RoboDK station: RoboDK.rdk

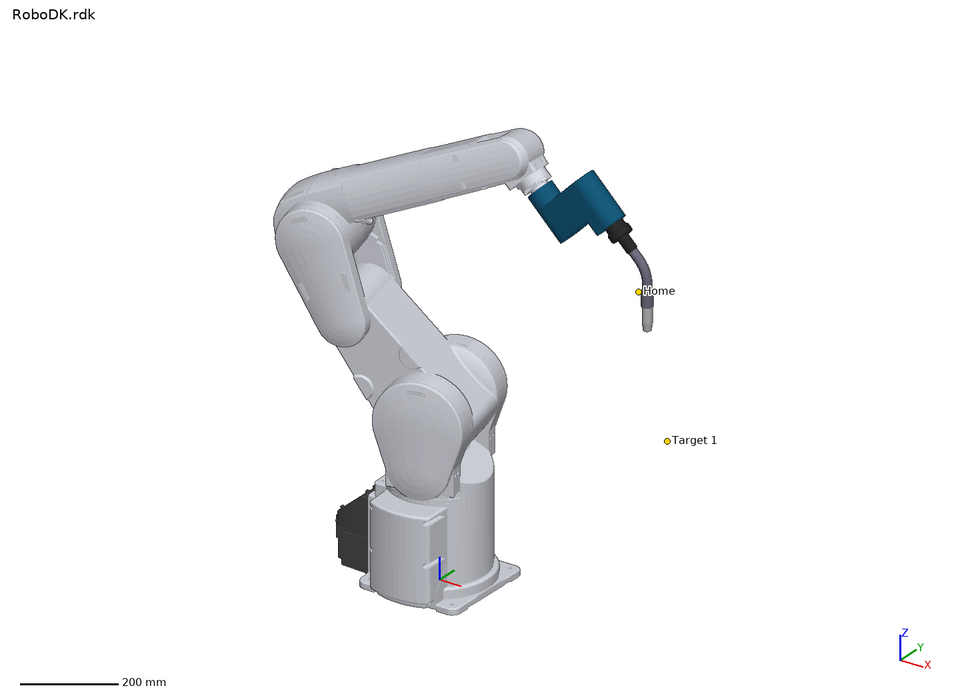
[picture v0: the station drawn from its stored meshes, robots at their saved joint values, targets as dots, program paths as lines]
Station 123. Poses are relative to the parent item; angles as X-Y-Z fixed-axis rotations.
  - frame Mitsubishi RV-7FL Base at (0, 0, 0) mm
    - robot Mitsubishi RV-7FL: 6 axes, payload 7 kg, reach 908 mm, repeatability 0.02 mm, weight 67 kg
        modified DH rows (alpha deg, a mm, theta deg, d mm): 0, 0, 0, 400; -90, 0, -90, 0; 0, 435, -90, 0; -90, 50, 0, 470; 90, 0, 0, 0; -90, 0, 180, 85
        joint limits [-240, -110, 0, -200, -120, -360] to [240, 130, 162, 200, 120, 360]; home [0, 0, 90, 0, 0, 0]; saved at [13.161, -34.303, 100.935, -9.903, 69.415, 12.901]
      - tool Weld gun, TCP at (-4, 0, 371.3) mm, rotated rx 0 ry 45 rz 0 deg, size 299.9 x 60 x 318.3 mm
    - target Home (Cartesian target) at (492.9, 0, 788.4) mm, rotated rx -180 ry 29.44 rz -180 deg; joints [0, -138.016, 114.252, 0, 39.328, 0] of Mitsubishi RV-7FL
    - target Target 1 (Cartesian target) at (564.87, 0, 471.83) mm, rotated rx -180 ry 0 rz -180 deg; joints [0, -116.511, 123.863, 0, 37.648, 0] of Mitsubishi RV-7FL
  - Python program Movement Imitation of Real-time Painting  (listed below)

--- Python program Movement Imitation of Real-time Painting  ---
from robolink import *    # API to communicate with RoboDK
from robodk import *      # robodk robotics toolbox

# Any interaction with RoboDK must be done through RDK:
RDK = Robolink()

# get the robot by name:
robot = RDK.Item('', ITEM_TYPE_ROBOT)

# get the home target and the welding targets:
home = RDK.Item('Home')
target = RDK.Item('Target 1')

# get the pose of the target (4x4 matrix representing position and orientation):
poseref = target.Pose()

# move the robot to home, then to the Target 1:
robot.MoveJ(home)
robot.MoveJ(target)

import socket

client = socket.socket()  # 默认是AF_INET、SOCK_STREAM
client.connect(('192.168.31.238',6868))
s = "hgdth"
client.send(s.encode("utf-8"))
xxx=0
yyy=0
mm=0
nn=0
judge="one"

while True:
    data = str(client.recv(1024))

    data=data[2:-1]
    data=data.split("#",5)

    xx = (int(data[1]) + int(data[3])) / 10 / 2

    yy=(int(data[0])+int(data[2]))/10/2

    label=data[4][2:-1]
    label=label.split(" ",2)[0]

    distence=int(float(data[5][:5])*1000)
    if distence!=0:

        if label=="fisted":

            if judge=="one":
                down1 =poseref*transl(xxx,yyy,-(150+50))
                robot.MoveL(down1)
                move1=poseref*transl(xx,yy,-(150+50))
                robot.MoveL(move1)
                judge="two"
                print("Moving")
            else:
                print("Not Moving")

        elif label=="brush-holding":

            if  400<distence and distence<800:
                up =poseref*transl(xxx,yyy,-(150+distence*6/80-10))
                print(-(150+distence*6/80-10))
                robot.MoveL(up)
                move=poseref*transl(xx,yy,-(150+distence*6/80-10))
                robot.MoveJ(move)
                judge="one"
            elif distence>=800:
                up =poseref*transl(xxx,yyy,-200)
                robot.MoveL(up)
                move=poseref*transl(xx,yy,-200)
                robot.MoveJ(move)
                judge="one"
            else:

                up =poseref*transl(xxx,yyy,-(150+distence*1/20))
                robot.MoveL(up)
                move=poseref*transl(xx,yy,-(150+distence*1/20))
                robot.MoveJ(move)
                judge="one"

        else:

            down =poseref*transl(xxx,yyy,-200)
            robot.MoveL(down)
            move=poseref*transl(xx,yy,-200)
            robot.MoveL(move)
            judge="one"

        xxx=xx
        yyy=yy
    else:
        print("Depth camera can't detect this point")
